(* IEC 61131-3 sources: stc/pkg/lexer/testdata, 4 files *)

(* ---- motor_control.st ---- *)
FUNCTION_BLOCK FB_Motor
VAR_INPUT
    Start : BOOL;
    Stop  : BOOL;
END_VAR
VAR_OUTPUT
    Running : BOOL;
END_VAR
IF Start AND NOT Stop THEN
    Running := TRUE;
END_IF;
END_FUNCTION_BLOCK

(* ---- oop_extensions.st ---- *)
INTERFACE IMotor
METHOD Start : BOOL
END_METHOD
END_INTERFACE

FUNCTION_BLOCK FB_Motor EXTENDS FB_Base IMPLEMENTS IMotor
VAR
    _running : BOOL;
END_VAR
METHOD PUBLIC Start : BOOL
    _running := TRUE;
    Start := _running;
END_METHOD
PROPERTY Running : BOOL
END_PROPERTY
END_FUNCTION_BLOCK

(* ---- pragmas.st ---- *)
{attribute 'qualified_only'}
FUNCTION_BLOCK FB_Global
VAR_GLOBAL
    {attribute 'symbol' := 'readwrite'}
    gCounter : INT;
END_VAR
END_FUNCTION_BLOCK

(* ---- typed_literals.st ---- *)
PROGRAM TypedLitTest
VAR
    a : INT := INT#42;
    b : REAL := REAL#3.14;
    c : INT := 16#FF;
    d : INT := 2#1010;
    e : TIME := T#5s;
    f : TIME := T#1h30m;
    g : DATE := D#2024-01-15;
    h : LREAL := LREAL#1.0E-5;
END_VAR
END_PROGRAM
